FUNCTION_BLOCK EC_SET_EVT (* Sets an event in- or output event of a FB instance (e.g. like an event sniffer) *)
  (* Standard: 61499-1; Classification: Reconfiguration; Function: Sets Event In-/Output; Type: Execution Control Service; Description: Copyright (c) 2012 Profactor GmbH This program and the accompanying materials are made available under the terms of the Eclipse Public License 2.0 which is available at https://www.eclipse.org/legal/epl-2.0/ SPDX-License-Identifier: EPL-2.0 *)
  (* Version 1.0, 2012-05-31, Gerhard Ebenhofer, Profactor GmbH *)
  (* Compiler Cpp GNU GCC >3.0 *)
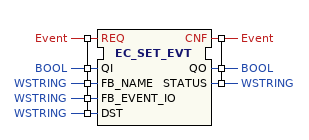
  EVENT_INPUT
    REQ WITH QI, DST, FB_NAME, FB_EVENT_IO; (* Service Request *)
  END_EVENT
  EVENT_OUTPUT
    CNF WITH QO, STATUS; (* Confirmation of Requested Service *)
  END_EVENT
  VAR_INPUT
    QI : BOOL; (* Event Input Qualifier *)
    FB_NAME : WSTRING; (* FunctionBlock instance name *)
    FB_EVENT_IO : WSTRING; (* event name *)
    DST : WSTRING; (* Destination where the event has to be set (Syntax: ResourceName) *)
  END_VAR
  VAR_OUTPUT
    QO : BOOL; (* Event Output Qualifier *)
    STATUS : WSTRING; (* Service Status: RDY, NO_SUCH_OBJECT, INVALID_STATE *)
  END_VAR
  SERVICE APPLICATION/RESOURCE (* Sets an event in- or output event of a FB instance (e.g. like an event sniffer) *)
    SEQUENCE normal_establishment
      APPLICATION.INIT+() -> APPLICATION.INITO+();
    END_SEQUENCE
    SEQUENCE unsuccessful_establishment
      APPLICATION.INIT+() -> APPLICATION.INITO-();
    END_SEQUENCE
    SEQUENCE request_confirm
      APPLICATION.REQ+() -> APPLICATION.CNF+();
    END_SEQUENCE
    SEQUENCE request_inhibited
      APPLICATION.REQ-() -> APPLICATION.CNF-();
    END_SEQUENCE
    SEQUENCE request_error
      APPLICATION.REQ+() -> APPLICATION.CNF-();
    END_SEQUENCE
    SEQUENCE application_initiated_termination
      APPLICATION.INIT-() -> APPLICATION.INITO-();
    END_SEQUENCE
    SEQUENCE resource_initiated_termination
      -> APPLICATION.INITO-();
    END_SEQUENCE
  END_SERVICE
END_FUNCTION_BLOCK
